{attribute 'linkalways'} 
{attribute 'no_explicit_call' := 'This FB is a CLASS and must be accessed using methods or properties'}
{attribute 'enable_dynamic_creation'}
FUNCTION_BLOCK RpcSynchronousResponseBuilder IMPLEMENTS I_RpcResponseBuilder;
VAR
	seralizer : I_Serializer;
	response : I_ServerResponse;
END_VAR

METHOD PUBLIC AddBase64 : I_RpcResponseBuilder
VAR_INPUT
	pBytes : POINTER TO BYTE;
	nBytes : DINT;
END_VAR
seralizer.AddBase64(pBytes, nBytes);
AddBase64 := THIS^;
END_METHOD

METHOD PUBLIC AddBool : I_RpcResponseBuilder
VAR_INPUT
	Value : BOOL;
END_VAR
seralizer.AddBool(Value);
AddBool := THIS^;
END_METHOD

METHOD PUBLIC AddBytesAsHex : I_RpcResponseBuilder
VAR_INPUT
	pBytes : POINTER TO BYTE;
	nBytes : DINT;
END_VAR
seralizer.AddBytesAsHex(pBytes, nBytes);
AddBytesAsHex := THIS^;
END_METHOD

METHOD PUBLIC AddDateTime : I_RpcResponseBuilder
VAR_INPUT
	Value : DATE_AND_TIME;
END_VAR
seralizer.AddDateTime(Value);
AddDateTime := THIS^;
END_METHOD

METHOD PUBLIC AddDcTime : I_RpcResponseBuilder
VAR_INPUT
	Value : DCTIME;
END_VAR
seralizer.AddDcTime(Value);
AddDcTime := THIS^;
END_METHOD

METHOD PUBLIC AddDint : I_RpcResponseBuilder
VAR_INPUT
	Value : DINT;
END_VAR
seralizer.AddDint(Value);
AddDint := THIS^;
END_METHOD

METHOD PUBLIC AddFileTime : I_RpcResponseBuilder
VAR_INPUT
	Value : FILETIME;
END_VAR
seralizer.AddFileTime(Value);
AddFileTime := THIS^;
END_METHOD

METHOD PUBLIC AddKey : I_RpcResponseBuilder
VAR_INPUT
	Key : T_MAXSTRING;
END_VAR
seralizer.AddKey(Key);
AddKey := THIS^;
END_METHOD

METHOD PUBLIC AddKeyBase64 : I_RpcResponseBuilder
VAR_INPUT
	Key : T_MAXSTRING;
	pBytes : POINTER TO BYTE;
	nBytes : DINT;
END_VAR
seralizer.AddKeyBase64(Key, pBytes, nBytes);
AddKeyBase64 := THIS^;
END_METHOD

METHOD PUBLIC AddKeyBool : I_RpcResponseBuilder
VAR_INPUT
	Key : T_MAXSTRING;
	Value : BOOL;
END_VAR
seralizer.AddKeyBool(Key,Value);
AddKeyBool := THIS^;
END_METHOD

METHOD PUBLIC AddKeyBytesAsHex : I_RpcResponseBuilder
VAR_INPUT
	Key : T_MAXSTRING;
	pBytes : POINTER TO BYTE;
	nBytes : DINT;
END_VAR
seralizer.AddKeyBytesAsHex(Key, pBytes, nBytes);
AddKeyBytesAsHex := THIS^;
END_METHOD

METHOD PUBLIC AddKeyDateTime : I_RpcResponseBuilder
VAR_INPUT
	Key : T_MAXSTRING;
	Value : DATE_AND_TIME;
END_VAR
seralizer.AddKeyDateTime(Key,Value);
AddKeyDateTime := THIS^;
END_METHOD

METHOD PUBLIC AddKeyDcTime : I_RpcResponseBuilder
VAR_INPUT
	Key : T_MAXSTRING;
	Value : DCTIME;
END_VAR
seralizer.AddKeyDcTime(Key,Value);
AddKeyDcTime := THIS^;
END_METHOD

METHOD PUBLIC AddKeyDint : I_RpcResponseBuilder
VAR_INPUT
	Key : T_MAXSTRING;
	Value : DINT;
END_VAR
seralizer.AddKeyDint(Key,Value);
AddKeyDint := THIS^;
END_METHOD

METHOD PUBLIC AddKeyFileTime : I_RpcResponseBuilder
VAR_INPUT
	Key : T_MAXSTRING;
	Value : FILETIME;
END_VAR
seralizer.AddKeyFileTime(Key,Value);
AddKeyFileTime := THIS^;
END_METHOD

METHOD PUBLIC AddKeyLint : I_RpcResponseBuilder
VAR_INPUT
	Key : T_MAXSTRING;
	Value : LINT;
END_VAR
seralizer.AddKeyLint(Key, Value);
AddKeyLint := THIS^;
END_METHOD

METHOD PUBLIC AddKeyLreal : I_RpcResponseBuilder
VAR_INPUT
	Key : T_MAXSTRING;
	Value : LREAL;
END_VAR
seralizer.AddKeyLreal(Key,Value);
AddKeyLreal := THIS^;
END_METHOD

METHOD PUBLIC AddKeyNull : I_RpcResponseBuilder
VAR_INPUT
	Key : T_MAXSTRING;
END_VAR
seralizer.AddKeyNull(Key);
AddKeyNull := THIS^;
END_METHOD

METHOD PUBLIC AddKeyReal : I_RpcResponseBuilder
VAR_INPUT
	Key : T_MAXSTRING;
	Value : REAL;
END_VAR
seralizer.AddKeyReal(Key, Value);
AddKeyReal := THIS^;
END_METHOD

METHOD PUBLIC AddKeyString : I_RpcResponseBuilder
VAR_INPUT
	Key : T_MAXSTRING;
	Value : T_MAXSTRING;
END_VAR
seralizer.AddKeyString(Key,Value);
AddKeyString := THIS^;
END_METHOD

METHOD PUBLIC AddKeyUdint : I_RpcResponseBuilder
VAR_INPUT
	Key : T_MAXSTRING;
	Value : UDINT;
END_VAR
seralizer.AddKeyUdint(Key, Value);
AddKeyUdint := THIS^;
END_METHOD

METHOD PUBLIC AddKeyUlint : I_RpcResponseBuilder
VAR_INPUT
	Key : T_MAXSTRING;
	Value : ULINT;
END_VAR
seralizer.AddKeyUlint(Key, Value);
AddKeyUlint := THIS^;
END_METHOD

METHOD PUBLIC AddLint : I_RpcResponseBuilder
VAR_INPUT
	Value : LINT;
END_VAR
seralizer.AddLint(Value);
AddLint := THIS^;
END_METHOD

METHOD PUBLIC AddLreal : I_RpcResponseBuilder
VAR_INPUT
	Value : LREAL;
END_VAR
seralizer.AddLreal(Value);
AddLreal := THIS^;
END_METHOD

METHOD PUBLIC AddNull : I_RpcResponseBuilder
VAR_INPUT
END_VAR
seralizer.AddNull();
AddNull := THIS^;
END_METHOD

METHOD PUBLIC AddReal : I_RpcResponseBuilder
VAR_INPUT
	Value : REAL;
END_VAR
seralizer.AddReal(Value);
AddReal := THIS^;
END_METHOD

METHOD PUBLIC AddString : I_RpcResponseBuilder
VAR_INPUT
	Value : T_MAXSTRING;
END_VAR
seralizer.AddString(Value);
AddString := THIS^;
END_METHOD

METHOD PUBLIC AddUdint : I_RpcResponseBuilder
VAR_INPUT
	Value : UDINT;
END_VAR
seralizer.AddUdint(Value);
AddUdint := THIS^;
END_METHOD

METHOD PUBLIC AddUlint : I_RpcResponseBuilder
VAR_INPUT
	Value : ULINT;
END_VAR
seralizer.AddUlint(Value);
AddUlint := THIS^;
END_METHOD

METHOD PUBLIC EndArray : I_RpcResponseBuilder
VAR_INPUT
END_VAR
seralizer.EndArray();
EndArray := THIS^;
END_METHOD

METHOD PUBLIC EndObject : I_RpcResponseBuilder
VAR_INPUT
END_VAR
seralizer.EndObject();
EndObject := THIS^;
END_METHOD

METHOD PUBLIC Initialize
VAR_INPUT
	Seralizer : I_Serializer;
	Response : I_ServerResponse;
END_VAR
THIS^.seralizer := Seralizer;
THIS^.response := Response;
END_METHOD

METHOD PUBLIC Reset
VAR_INPUT
END_VAR
seralizer.Reset();
END_METHOD

METHOD PUBLIC Send
VAR_INPUT
END_VAR
VAR
	jsonSize : UDINT;
	pJsonString : POINTER TO STRING;
END_VAR
jsonSize := seralizer.GetSeralizedDataLength();

IF jsonSize = 0 THEN
	response.Error('RPC Handler returned invalid object');
	RETURN;
END_IF

pJsonString := __NEW(BYTE, jsonSize);

IF NOT seralizer.TryGetSerialziedData(pJsonString, jsonSize) THEN
	response.Error('RPC Handler unable to get serialized data');
	__DELETE(pJsonString);
	RETURN;
END_IF

response.SuccessWithPayload(pJsonString, jsonSize);
__DELETE(pJsonString);
END_METHOD

METHOD PUBLIC StartArray : I_RpcResponseBuilder
VAR_INPUT
END_VAR
seralizer.StartArray();
StartArray := THIS^;
END_METHOD

METHOD PUBLIC StartObject : I_RpcResponseBuilder
VAR_INPUT
END_VAR
seralizer.StartObject();
StartObject := THIS^;
END_METHOD

END_FUNCTION_BLOCK

(* stored: Version 1.1.0.1, ProductVersion 3.1.4024.12
   POU RpcSynchronousResponseBuilder: Id {65e3981c-03d0-4a54-8803-bd1abcc522d0}, SpecialFunc None
   Method AddBase64: Id {fd7e585a-cce0-4c64-af14-22c6b6ebcff4}
   Method AddBool: Id {9cf935fe-ea6b-4559-92e5-825b2ad74d57}
   Method AddBytesAsHex: Id {8dc6fe8e-09fe-4bb7-961c-e7574b8056a6}
   Method AddDateTime: Id {5ca1875f-d970-48d0-808b-aa20c0735d1d}
   Method AddDcTime: Id {ed24a5c9-6cd6-40cb-8b01-cb43dfc42c32}
   Method AddDint: Id {3e9af678-a30a-4489-9f9c-a783b697ead9}
   Method AddFileTime: Id {ccdaacb6-778e-471a-a1f8-eadfba8d565f}
   Method AddKey: Id {49f8803f-9f30-4444-aa98-e3a1b92c2f3b}
   Method AddKeyBase64: Id {a1fd7d62-b87b-439b-8ef6-28ae6bf17314}
   Method AddKeyBool: Id {2255d073-79dc-4ca9-9ac3-9ca57a878d41}
   Method AddKeyBytesAsHex: Id {7f583573-96ff-4a08-9f47-e90e1f4600cc}
   Method AddKeyDateTime: Id {6999b15d-1935-4bf9-948b-10257fae564f}
   Method AddKeyDcTime: Id {2b8fe65c-7296-4a9a-9229-75acaedded87}
   Method AddKeyDint: Id {8e6f462d-5aa7-40e4-83cc-529d89661656}
   Method AddKeyFileTime: Id {8b208ad8-8241-4d19-9478-3ea16932d2f0}
   Method AddKeyLint: Id {e5ab8a1a-d54f-4ef1-adde-3f913acf65cc}
   Method AddKeyLreal: Id {b4d707d1-0708-4b5d-9422-0da022815c1e}
   Method AddKeyNull: Id {7272ab36-8361-46fd-a92d-eaa99797f0ee}
   Method AddKeyReal: Id {bc4302fb-f8fc-4296-b4f0-fb3a08dab09d}
   Method AddKeyString: Id {71953099-587d-4c30-8596-bf3f0daa6a28}
   Method AddKeyUdint: Id {ee7f493e-d839-4a94-8f78-9303e339398c}
   Method AddKeyUlint: Id {45897fdc-ccb7-4ee5-a899-bb105ab47ce6}
   Method AddLint: Id {b66b044c-ce05-45bc-9dbc-9029bc5d04cc}
   Method AddLreal: Id {d508304e-c47d-4779-8cc4-47646b2f5a1a}
   Method AddNull: Id {722b0750-c8b4-4b8f-b2dc-2b028e902b46}
   Method AddReal: Id {48daf22f-962c-45e0-9ef7-11fb9eb97738}
   Method AddString: Id {e096eef1-b9eb-4414-b232-89956b2fb45c}
   Method AddUdint: Id {21c16e77-2eb3-4195-ad96-b116be705966}
   Method AddUlint: Id {df59dcc9-72c7-425f-8aee-110d5a30f2d5}
   Method EndArray: Id {7cb322ba-ea6d-4e83-9746-5a973615438b}
   Method EndObject: Id {59935545-1eb5-4676-88bb-17cda55c7ba6}
   Method Initialize: Id {974d68b6-add8-4295-a69d-4e8fff7f96df}
   Method Reset: Id {f7bf4797-65b3-47a1-94cd-15ee2a80f58b}
   Method Send: Id {9bd68d42-b7b6-4370-88c0-e2cc10c5fabe}
   Method StartArray: Id {f6863fbc-98ac-4960-93a2-baf047f5f81e}
   Method StartObject: Id {a7ced10e-2813-420e-8f2a-e223701ed045} *)
